FUNCTION Convert_SINT_TO_DATE : Hresult
VAR_INPUT
	in : SINT;
	out : REFERENCE TO DATE;
END_VAR
VAR
	converted : DATE;
END_VAR
VAR CONSTANT
	INCOMPATIBLE : HRESULT := 16#9811070E;
END_VAR

converted := SINT_TO_DATE(in);

IF (DATE_TO_SINT(converted) <> in) THEN
	Convert_SINT_TO_DATE := INCOMPATIBLE;
	RETURN;
END_IF

out := converted;

END_FUNCTION

(* stored: Version 1.1.0.1, ProductVersion 3.1.4024.12
   POU Convert_SINT_TO_DATE: Id {fe73700d-82ed-478c-b11f-0ce97aa19939}, SpecialFunc None *)
